FUNCTION F_DeviceTwin_GetSubscriberTopicDesired : STRING
VAR_INPUT
END_VAR
VAR
END_VAR

F_DeviceTwin_GetSubscriberTopicDesired := '$$iothub/twin/PATCH/properties/desired/#';

END_FUNCTION

(* stored: Version 1.1.0.1, ProductVersion 3.1.4022.3
   POU F_DeviceTwin_GetSubscriberTopicDesired: Id {864463c2-3abb-4edf-9f72-90da71418645}, SpecialFunc None *)
